FUNCTION_BLOCK EL2784
VAR
	{attribute addProperty Name "WcState"}
	_wcState : WcStateBase;
	{attribute addProperty Name "Info data"}
	_infoData : InfoDataBase;
	_io : EL2xx4_Data;
END_VAR

PROPERTY IO : REFERENCE TO EL2xx4_Data
GET
IO REF= _io;
END_GET
END_PROPERTY

PROPERTY WcState : REFERENCE TO WcStateBase
GET
WcState REF= _wcState;
END_GET
END_PROPERTY

END_FUNCTION_BLOCK

(* stored: Version 1.1.0.1, ProductVersion 3.1.4024.9
   POU EL2784: Id {9f0d08d9-eebe-0578-1a70-81276ab5339c}, SpecialFunc None
   Property IO: Id {a8408cab-228e-05b8-0ef3-ba20e1cc4a99}
   Get Get: Id {e3f111fe-fb42-034b-1a5d-fa4187f31aaf}
   Property WcState: Id {d48a82bc-2a4d-0790-3827-80e9945180e1}
   Get Get: Id {368bc1ab-c777-042b-34eb-c7f456b5cde6} *)
